KUKA KRL program: DESPA - KR 470-2 PA.src, DESPA - KR 470-2 PA.dat

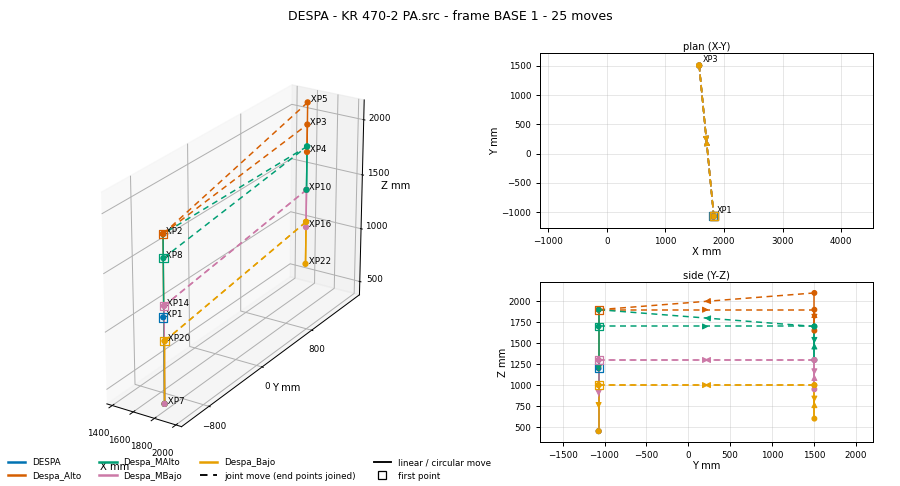
[picture p0: tool path of DESPA - KR 470-2 PA.src in frame BASE 1, 25 of 25 moves have a stored position in this frame; points joined in program order, loops and branches not executed]
--- DESPA - KR 470-2 PA.src ---
&ACCESS RVP
&REL 5
&PARAM TEMPLATE = C:\KRC\ROBOTER\TEMPLATE\vorgabe
&PARAM EDITMASK = *
DEF DESPA - KR 470-2 PA( )
;FOLD INI;%{PE}%V3.2.0,%MKUKATPBASIS,%CINIT,%VCOMMON,%P
;FOLD BAS INI;%{E}%V3.2.0,%MKUKATPBASIS,%CINIT,%VINIT,%P
GLOBAL INTERRUPT DECL 3 WHEN $STOPMESS==TRUE DO IR_STOPM ( )
INTERRUPT ON 3
BAS (#INITMOV,0 )
;ENDFOLD (BAS INI)
;FOLD A20 INI;%{E}%V3.2.0,%MKUKATPA20,%CINIT,%VINIT,%P
IF ARC20==TRUE THEN
A20 (ARC_INI)
INTERRUPT DECL 6 WHEN $CYCFLAG[3]==FALSE DO A20(TECH_STOP2)
ENDIF
;ENDFOLD (A20 INI)
;FOLD A10 INI;%{E}%V3.2.0,%MKUKATPARC,%CINIT,%VINIT,%P
IF A10_OPTION==#ACTIVE THEN
INTERRUPT DECL 4 WHEN $CYCFLAG[2]==FALSE DO A10 (#APPL_ERROR)
INTERRUPT DECL 7 WHEN A_ARC_SWI==#ACTIVE DO A10 (#ARC_SEAM)
INTERRUPT DECL 5 WHEN A_FLY_ARC==TRUE DO A10 (#HPU_ARC)
INTERRUPT  ON 5
A10_INI ( )
ENDIF
;ENDFOLD (A10 INI)
;FOLD GRIPPER INI;%{E}%V3.2.0,%MKUKATPGRIPPER,%CINIT,%VINIT,%P
USER_GRP(0,DUMMY,DUMMY,GDEFAULT)
;ENDFOLD (GRIPPER INI)
;FOLD SPOT INI;%{E}%V3.2.0,%MKUKATPSPOT,%CINIT,%VINIT,%P
USERSPOT(#INIT)
;ENDFOLD (SPOT INI)
;FOLD TOUCHSENSE INI;%{E}%V3.2.0,%MKUKATPTS,%CINIT,%VINIT,%P
IF H70_OPTION THEN
INTERRUPT DECL 15 WHEN $MEAS_PULSE[TOUCH_I[TOUCH_ACTIVE].IN_NR] DO H70 (6,CD0 )
INTERRUPT DECL 16 WHEN $ZERO_MOVE DO H70 (7,CD0 )
INTERRUPT DECL 17 WHEN $TECHPAR_C[FG_TOUCH,8]>0.5 DO H70 (8,CD0)
H70 (1,CD0 )
ENDIF
;ENDFOLD (TOUCHSENSE INI)
;FOLD USER INI;%{E}%V3.2.0,%MKUKATPUSER,%CINIT,%VINIT,%P
;Make your modifications here
;ENDFOLD (USER INI)
;ENDFOLD (INI)

; Layout : C:\Users\Albert\Desktop\Proy_Final\Final_V2\FINAL_V2.vcm
; Robot : KR 180 PA #3
; BASE_DATA[1] = {x 0,y 0,z 0,a 0,b 0,c 0}
; TOOL_DATA[1] = {x 0,y 0,z 0,a 0,b 0,c 0}
Despa_Alto()
;FOLD WAIT Time= 0.5 sec;%{PE}%R 4.1.6,%MKUKATPBASIS,%CWAIT,%VWAIT,%P 2:0.5
WAIT SEC 0.5
;ENDFOLD
Despa_MAlto()
;FOLD WAIT Time= 1 sec;%{PE}%R 4.1.6,%MKUKATPBASIS,%CWAIT,%VWAIT,%P 2:1
WAIT SEC 1
;ENDFOLD
Despa_MBajo()
;FOLD WAIT Time= 1 sec;%{PE}%R 4.1.6,%MKUKATPBASIS,%CWAIT,%VWAIT,%P 2:1
WAIT SEC 1
;ENDFOLD
Despa_Bajo()
;FOLD WAIT Time= 1 sec;%{PE}%R 4.1.6,%MKUKATPBASIS,%CWAIT,%VWAIT,%P 2:1
WAIT SEC 1
;ENDFOLD
;FOLD LIN P1  Vel= 2 m/s CPDAT1 Tool[1] Base[1];%{PE}%R 4.1.6,%MKUKATPBASIS,%CMOVE,%VLIN,%P 1:LIN, 2:P1, 3:, 5:2, 7:CPDAT1
$BWDSTART = FALSE
LDAT_ACT=LCPDAT1
BAS(#CP_DAT)
FDAT_ACT=FP1
BAS(#FRAMES)
BAS(#VEL_CP,2)
LIN XP1
;ENDFOLD
END

DEF Despa_Alto()
;FOLD PTP P2  Vel= 100 % PDAT1 Tool[1] Base[1];%{PE}%R 4.1.6,%MKUKATPBASIS,%CMOVE,%VPTP,%P 1:PTP, 2:P2, 3:, 5:100, 7:PDAT1
$BWDSTART = FALSE
PDAT_ACT=PPDAT1
BAS(#PTP_DAT)
FDAT_ACT=FP2
BAS(#FRAMES)
BAS(#VEL_PTP,100)
PTP XP2
;ENDFOLD
;FOLD PTP P3  Vel= 100 % PDAT2 Tool[1] Base[1];%{PE}%R 4.1.6,%MKUKATPBASIS,%CMOVE,%VPTP,%P 1:PTP, 2:P3, 3:, 5:100, 7:PDAT2
$BWDSTART = FALSE
PDAT_ACT=PPDAT2
BAS(#PTP_DAT)
FDAT_ACT=FP3
BAS(#FRAMES)
BAS(#VEL_PTP,100)
PTP XP3
;ENDFOLD
;FOLD LIN P4  Vel= 2 m/s CPDAT2 Tool[1] Base[1];%{PE}%R 4.1.6,%MKUKATPBASIS,%CMOVE,%VLIN,%P 1:LIN, 2:P4, 3:, 5:2, 7:CPDAT2
$BWDSTART = FALSE
LDAT_ACT=LCPDAT2
BAS(#CP_DAT)
FDAT_ACT=FP4
BAS(#FRAMES)
BAS(#VEL_CP,2)
LIN XP4
;ENDFOLD
;FOLD LIN P5  Vel= 2 m/s CPDAT3 Tool[1] Base[1];%{PE}%R 4.1.6,%MKUKATPBASIS,%CMOVE,%VLIN,%P 1:LIN, 2:P5, 3:, 5:2, 7:CPDAT3
$BWDSTART = FALSE
LDAT_ACT=LCPDAT3
BAS(#CP_DAT)
FDAT_ACT=FP5
BAS(#FRAMES)
BAS(#VEL_CP,2)
LIN XP5
;ENDFOLD
;FOLD PTP P6  Vel= 100 % PDAT3 Tool[1] Base[1];%{PE}%R 4.1.6,%MKUKATPBASIS,%CMOVE,%VPTP,%P 1:PTP, 2:P6, 3:, 5:100, 7:PDAT3
$BWDSTART = FALSE
PDAT_ACT=PPDAT3
BAS(#PTP_DAT)
FDAT_ACT=FP6
BAS(#FRAMES)
BAS(#VEL_PTP,100)
PTP XP6
;ENDFOLD
;FOLD LIN P7  Vel= 2 m/s CPDAT4 Tool[1] Base[1];%{PE}%R 4.1.6,%MKUKATPBASIS,%CMOVE,%VLIN,%P 1:LIN, 2:P7, 3:, 5:2, 7:CPDAT4
$BWDSTART = FALSE
LDAT_ACT=LCPDAT4
BAS(#CP_DAT)
FDAT_ACT=FP7
BAS(#FRAMES)
BAS(#VEL_CP,2)
LIN XP7
;ENDFOLD
END

DEF Despa_MAlto()
;FOLD PTP P8  Vel= 100 % PDAT4 Tool[1] Base[1];%{PE}%R 4.1.6,%MKUKATPBASIS,%CMOVE,%VPTP,%P 1:PTP, 2:P8, 3:, 5:100, 7:PDAT4
$BWDSTART = FALSE
PDAT_ACT=PPDAT4
BAS(#PTP_DAT)
FDAT_ACT=FP8
BAS(#FRAMES)
BAS(#VEL_PTP,100)
PTP XP8
;ENDFOLD
;FOLD PTP P9  Vel= 100 % PDAT5 Tool[1] Base[1];%{PE}%R 4.1.6,%MKUKATPBASIS,%CMOVE,%VPTP,%P 1:PTP, 2:P9, 3:, 5:100, 7:PDAT5
$BWDSTART = FALSE
PDAT_ACT=PPDAT5
BAS(#PTP_DAT)
FDAT_ACT=FP9
BAS(#FRAMES)
BAS(#VEL_PTP,100)
PTP XP9
;ENDFOLD
;FOLD LIN P10  Vel= 2 m/s CPDAT5 Tool[1] Base[1];%{PE}%R 4.1.6,%MKUKATPBASIS,%CMOVE,%VLIN,%P 1:LIN, 2:P10, 3:, 5:2, 7:CPDAT5
$BWDSTART = FALSE
LDAT_ACT=LCPDAT5
BAS(#CP_DAT)
FDAT_ACT=FP10
BAS(#FRAMES)
BAS(#VEL_CP,2)
LIN XP10
;ENDFOLD
;FOLD LIN P11  Vel= 2 m/s CPDAT6 Tool[1] Base[1];%{PE}%R 4.1.6,%MKUKATPBASIS,%CMOVE,%VLIN,%P 1:LIN, 2:P11, 3:, 5:2, 7:CPDAT6
$BWDSTART = FALSE
LDAT_ACT=LCPDAT6
BAS(#CP_DAT)
FDAT_ACT=FP11
BAS(#FRAMES)
BAS(#VEL_CP,2)
LIN XP11
;ENDFOLD
;FOLD PTP P12  Vel= 100 % PDAT6 Tool[1] Base[1];%{PE}%R 4.1.6,%MKUKATPBASIS,%CMOVE,%VPTP,%P 1:PTP, 2:P12, 3:, 5:100, 7:PDAT6
$BWDSTART = FALSE
PDAT_ACT=PPDAT6
BAS(#PTP_DAT)
FDAT_ACT=FP12
BAS(#FRAMES)
BAS(#VEL_PTP,100)
PTP XP12
;ENDFOLD
;FOLD LIN P13  Vel= 2 m/s CPDAT7 Tool[1] Base[1];%{PE}%R 4.1.6,%MKUKATPBASIS,%CMOVE,%VLIN,%P 1:LIN, 2:P13, 3:, 5:2, 7:CPDAT7
$BWDSTART = FALSE
LDAT_ACT=LCPDAT7
BAS(#CP_DAT)
FDAT_ACT=FP13
BAS(#FRAMES)
BAS(#VEL_CP,2)
LIN XP13
;ENDFOLD
END

DEF Despa_MBajo()
;FOLD PTP P14  Vel= 100 % PDAT7 Tool[1] Base[1];%{PE}%R 4.1.6,%MKUKATPBASIS,%CMOVE,%VPTP,%P 1:PTP, 2:P14, 3:, 5:100, 7:PDAT7
$BWDSTART = FALSE
PDAT_ACT=PPDAT7
BAS(#PTP_DAT)
FDAT_ACT=FP14
BAS(#FRAMES)
BAS(#VEL_PTP,100)
PTP XP14
;ENDFOLD
;FOLD PTP P15  Vel= 100 % PDAT8 Tool[1] Base[1];%{PE}%R 4.1.6,%MKUKATPBASIS,%CMOVE,%VPTP,%P 1:PTP, 2:P15, 3:, 5:100, 7:PDAT8
$BWDSTART = FALSE
PDAT_ACT=PPDAT8
BAS(#PTP_DAT)
FDAT_ACT=FP15
BAS(#FRAMES)
BAS(#VEL_PTP,100)
PTP XP15
;ENDFOLD
;FOLD LIN P16  Vel= 2 m/s CPDAT8 Tool[1] Base[1];%{PE}%R 4.1.6,%MKUKATPBASIS,%CMOVE,%VLIN,%P 1:LIN, 2:P16, 3:, 5:2, 7:CPDAT8
$BWDSTART = FALSE
LDAT_ACT=LCPDAT8
BAS(#CP_DAT)
FDAT_ACT=FP16
BAS(#FRAMES)
BAS(#VEL_CP,2)
LIN XP16
;ENDFOLD
;FOLD LIN P17  Vel= 2 m/s CPDAT9 Tool[1] Base[1];%{PE}%R 4.1.6,%MKUKATPBASIS,%CMOVE,%VLIN,%P 1:LIN, 2:P17, 3:, 5:2, 7:CPDAT9
$BWDSTART = FALSE
LDAT_ACT=LCPDAT9
BAS(#CP_DAT)
FDAT_ACT=FP17
BAS(#FRAMES)
BAS(#VEL_CP,2)
LIN XP17
;ENDFOLD
;FOLD PTP P18  Vel= 100 % PDAT9 Tool[1] Base[1];%{PE}%R 4.1.6,%MKUKATPBASIS,%CMOVE,%VPTP,%P 1:PTP, 2:P18, 3:, 5:100, 7:PDAT9
$BWDSTART = FALSE
PDAT_ACT=PPDAT9
BAS(#PTP_DAT)
FDAT_ACT=FP18
BAS(#FRAMES)
BAS(#VEL_PTP,100)
PTP XP18
;ENDFOLD
;FOLD LIN P19  Vel= 2 m/s CPDAT10 Tool[1] Base[1];%{PE}%R 4.1.6,%MKUKATPBASIS,%CMOVE,%VLIN,%P 1:LIN, 2:P19, 3:, 5:2, 7:CPDAT10
$BWDSTART = FALSE
LDAT_ACT=LCPDAT10
BAS(#CP_DAT)
FDAT_ACT=FP19
BAS(#FRAMES)
BAS(#VEL_CP,2)
LIN XP19
;ENDFOLD
END

DEF Despa_Bajo()
;FOLD PTP P20  Vel= 100 % PDAT10 Tool[1] Base[1];%{PE}%R 4.1.6,%MKUKATPBASIS,%CMOVE,%VPTP,%P 1:PTP, 2:P20, 3:, 5:100, 7:PDAT10
$BWDSTART = FALSE
PDAT_ACT=PPDAT10
BAS(#PTP_DAT)
FDAT_ACT=FP20
BAS(#FRAMES)
BAS(#VEL_PTP,100)
PTP XP20
;ENDFOLD
;FOLD PTP P21  Vel= 100 % PDAT11 Tool[1] Base[1];%{PE}%R 4.1.6,%MKUKATPBASIS,%CMOVE,%VPTP,%P 1:PTP, 2:P21, 3:, 5:100, 7:PDAT11
$BWDSTART = FALSE
PDAT_ACT=PPDAT11
BAS(#PTP_DAT)
FDAT_ACT=FP21
BAS(#FRAMES)
BAS(#VEL_PTP,100)
PTP XP21
;ENDFOLD
;FOLD LIN P22  Vel= 2 m/s CPDAT11 Tool[1] Base[1];%{PE}%R 4.1.6,%MKUKATPBASIS,%CMOVE,%VLIN,%P 1:LIN, 2:P22, 3:, 5:2, 7:CPDAT11
$BWDSTART = FALSE
LDAT_ACT=LCPDAT11
BAS(#CP_DAT)
FDAT_ACT=FP22
BAS(#FRAMES)
BAS(#VEL_CP,2)
LIN XP22
;ENDFOLD
;FOLD LIN P23  Vel= 2 m/s CPDAT12 Tool[1] Base[1];%{PE}%R 4.1.6,%MKUKATPBASIS,%CMOVE,%VLIN,%P 1:LIN, 2:P23, 3:, 5:2, 7:CPDAT12
$BWDSTART = FALSE
LDAT_ACT=LCPDAT12
BAS(#CP_DAT)
FDAT_ACT=FP23
BAS(#FRAMES)
BAS(#VEL_CP,2)
LIN XP23
;ENDFOLD
;FOLD PTP P24  Vel= 100 % PDAT12 Tool[1] Base[1];%{PE}%R 4.1.6,%MKUKATPBASIS,%CMOVE,%VPTP,%P 1:PTP, 2:P24, 3:, 5:100, 7:PDAT12
$BWDSTART = FALSE
PDAT_ACT=PPDAT12
BAS(#PTP_DAT)
FDAT_ACT=FP24
BAS(#FRAMES)
BAS(#VEL_PTP,100)
PTP XP24
;ENDFOLD
;FOLD LIN P25  Vel= 2 m/s CPDAT13 Tool[1] Base[1];%{PE}%R 4.1.6,%MKUKATPBASIS,%CMOVE,%VLIN,%P 1:LIN, 2:P25, 3:, 5:2, 7:CPDAT13
$BWDSTART = FALSE
LDAT_ACT=LCPDAT13
BAS(#CP_DAT)
FDAT_ACT=FP25
BAS(#FRAMES)
BAS(#VEL_CP,2)
LIN XP25
;ENDFOLD
END

--- DESPA - KR 470-2 PA.dat ---
&ACCESS RVP
&REL 5
&PARAM TEMPLATE = C:\KRC\ROBOTER\TEMPLATE\vorgabe
&PARAM EDITMASK = *
DEFDAT  despa - kr 470-2 pa
;FOLD EXTERNAL DECLARATIONS;%{PE}%V3.2.0,%MKUKATPBASIS,%CEXT,%VCOMMON,%P
;FOLD BAS EXT;%{PE}%V3.2.0,%MKUKATPBASIS,%CEXT,%VEXT,%P
EXT  BAS (BAS_COMMAND  :IN,REAL  :IN )
DECL INT SUCCESS
;ENDFOLD
;FOLD A10 EXT;%{E}%V3.2.0,%MKUKATPARC,%CEXT,%VEXT,%P
EXT  A10 (A_CMD_T  :IN,A_STRT_T  :IN,A_WELD_T  :IN,A_END_T  :IN,INT  :IN )
;ENDFOLD
;FOLD A20 EXT;%{E}%V3.2.0,%MKUKATPA20,%CEXT,%VEXT,%P
EXT  A20 (INT  :IN,WELD_ST  :IN,WELD_FI  :IN,INT  :IN )
;ENDFOLD
;FOLD GRIPPER EXT;%{E}%V3.2.0,%MKUKATPGRIPPER,%CEXT,%VEXT,%P
EXT  H50 (INT  :IN,INT  :IN,INT  :IN,GRP_TYP  :IN )
;ENDFOLD
;FOLD SPOT EXT;%{E}%V3.2.0,%MKUKATPSPOT,%CEXT,%VEXT,%P
EXT  USERSPOT (S_COMMAND  :IN,SPOT_TYPE  :IN )
;ENDFOLD
;FOLD TOUCHSENSE EXT;%{E}%V3.2.0,%MKUKATPTS,%CEXT,%VEXT,%P
EXT  H70 (INT  :IN,SRCH_TYP_2  :OUT,E6POS  :IN,SRCH_TYP_3  :IN,SRCH_TYP_2  :IN,SRCH_TYP_2  :IN,SRCH_TYP_2  :IN,SRCH_TYP_2  :IN,SRCH_TYP_2  :IN,INT  :IN )
;ENDFOLD
;FOLD USER EXT;%{E}%V3.2.0,%MKUKATPUSER,%CEXT,%VEXT,%P
;Make here your modifications
;ENDFOLD
;ENDFOLD

DECL E6POS XP1={x 1815.4,y -1070.28,z 1200,a -90,b 0,c -180,s 2,t 2,e1 0,e2 0,e3 0,e4 0,e5 0,e6 0}
DECL FDAT FP1={TOOL_NO 1,BASE_NO 1,IPO_FRAME #BASE}
DECL LDAT LCPDAT1={VEL 2.0,ACC 100.0,APO_DIST 100.0,APO_FAC 50.0}
DECL E6POS XP2={x 1825.4,y -1070.28,z 1900,a 90,b -180,c 0,s 2,t 2,e1 0,e2 0,e3 0,e4 0,e5 0,e6 0}
DECL FDAT FP2={TOOL_NO 1,BASE_NO 1,IPO_FRAME #BASE}
DECL PDAT PPDAT1={VEL 100.0,ACC 100.0,APO_DIST 100.0}
DECL E6POS XP3={x 1575.4,y 1504.72,z 1900,a 0,b 180,c 0,s 2,t 35,e1 0,e2 0,e3 0,e4 0,e5 0,e6 0}
DECL FDAT FP3={TOOL_NO 1,BASE_NO 1,IPO_FRAME #BASE}
DECL PDAT PPDAT2={VEL 100.0,ACC 100.0,APO_DIST 100.0}
DECL E6POS XP4={x 1575.4,y 1504.72,z 1650,a 0,b 180,c 0,s 2,t 35,e1 0,e2 0,e3 0,e4 0,e5 0,e6 0}
DECL FDAT FP4={TOOL_NO 1,BASE_NO 1,IPO_FRAME #BASE}
DECL LDAT LCPDAT2={VEL 2.0,ACC 100.0,APO_DIST 100.0,APO_FAC 50.0}
DECL E6POS XP5={x 1575.4,y 1504.72,z 2100,a 0,b 180,c 0,s 2,t 35,e1 0,e2 0,e3 0,e4 0,e5 0,e6 0}
DECL FDAT FP5={TOOL_NO 1,BASE_NO 1,IPO_FRAME #BASE}
DECL LDAT LCPDAT3={VEL 2.0,ACC 100.0,APO_DIST 100.0,APO_FAC 50.0}
DECL E6POS XP6={x 1825.4,y -1070.28,z 1900,a 90,b 180,c 0,s 2,t 2,e1 0,e2 0,e3 0,e4 0,e5 0,e6 0}
DECL FDAT FP6={TOOL_NO 1,BASE_NO 1,IPO_FRAME #BASE}
DECL PDAT PPDAT3={VEL 100.0,ACC 100.0,APO_DIST 100.0}
DECL E6POS XP7={x 1815.4,y -1070.28,z 450,a -90,b 0,c 180,s 2,t 2,e1 0,e2 0,e3 0,e4 0,e5 0,e6 0}
DECL FDAT FP7={TOOL_NO 1,BASE_NO 1,IPO_FRAME #BASE}
DECL LDAT LCPDAT4={VEL 2.0,ACC 100.0,APO_DIST 100.0,APO_FAC 50.0}
DECL E6POS XP8={x 1825.4,y -1070.28,z 1700,a 90,b -180,c 0,s 2,t 2,e1 0,e2 0,e3 0,e4 0,e5 0,e6 0}
DECL FDAT FP8={TOOL_NO 1,BASE_NO 1,IPO_FRAME #BASE}
DECL PDAT PPDAT4={VEL 100.0,ACC 100.0,APO_DIST 100.0}
DECL E6POS XP9={x 1575.4,y 1504.72,z 1700,a 0,b 180,c 0,s 2,t 35,e1 0,e2 0,e3 0,e4 0,e5 0,e6 0}
DECL FDAT FP9={TOOL_NO 1,BASE_NO 1,IPO_FRAME #BASE}
DECL PDAT PPDAT5={VEL 100.0,ACC 100.0,APO_DIST 100.0}
DECL E6POS XP10={x 1575.4,y 1504.72,z 1300,a 0,b 180,c 0,s 2,t 35,e1 0,e2 0,e3 0,e4 0,e5 0,e6 0}
DECL FDAT FP10={TOOL_NO 1,BASE_NO 1,IPO_FRAME #BASE}
DECL LDAT LCPDAT5={VEL 2.0,ACC 100.0,APO_DIST 100.0,APO_FAC 50.0}
DECL E6POS XP11={x 1575.4,y 1504.72,z 1700,a 0,b 180,c 0,s 2,t 35,e1 0,e2 0,e3 0,e4 0,e5 0,e6 0}
DECL FDAT FP11={TOOL_NO 1,BASE_NO 1,IPO_FRAME #BASE}
DECL LDAT LCPDAT6={VEL 2.0,ACC 100.0,APO_DIST 100.0,APO_FAC 50.0}
DECL E6POS XP12={x 1825.4,y -1070.28,z 1900,a 90,b 180,c 0,s 2,t 2,e1 0,e2 0,e3 0,e4 0,e5 0,e6 0}
DECL FDAT FP12={TOOL_NO 1,BASE_NO 1,IPO_FRAME #BASE}
DECL PDAT PPDAT6={VEL 100.0,ACC 100.0,APO_DIST 100.0}
DECL E6POS XP13={x 1815.4,y -1070.28,z 450,a -90,b 0,c -180,s 2,t 2,e1 0,e2 0,e3 0,e4 0,e5 0,e6 0}
DECL FDAT FP13={TOOL_NO 1,BASE_NO 1,IPO_FRAME #BASE}
DECL LDAT LCPDAT7={VEL 2.0,ACC 100.0,APO_DIST 100.0,APO_FAC 50.0}
DECL E6POS XP14={x 1825.4,y -1070.28,z 1300,a 90,b -180,c 0,s 2,t 2,e1 0,e2 0,e3 0,e4 0,e5 0,e6 0}
DECL FDAT FP14={TOOL_NO 1,BASE_NO 1,IPO_FRAME #BASE}
DECL PDAT PPDAT7={VEL 100.0,ACC 100.0,APO_DIST 100.0}
DECL E6POS XP15={x 1575.4,y 1504.72,z 1300,a 0,b 180,c 0,s 2,t 35,e1 0,e2 0,e3 0,e4 0,e5 0,e6 0}
DECL FDAT FP15={TOOL_NO 1,BASE_NO 1,IPO_FRAME #BASE}
DECL PDAT PPDAT8={VEL 100.0,ACC 100.0,APO_DIST 100.0}
DECL E6POS XP16={x 1575.4,y 1504.72,z 950,a 0,b 180,c 0,s 2,t 35,e1 0,e2 0,e3 0,e4 0,e5 0,e6 0}
DECL FDAT FP16={TOOL_NO 1,BASE_NO 1,IPO_FRAME #BASE}
DECL LDAT LCPDAT8={VEL 2.0,ACC 100.0,APO_DIST 100.0,APO_FAC 50.0}
DECL E6POS XP17={x 1575.4,y 1504.72,z 1300,a 0,b 180,c 0,s 2,t 35,e1 0,e2 0,e3 0,e4 0,e5 0,e6 0}
DECL FDAT FP17={TOOL_NO 1,BASE_NO 1,IPO_FRAME #BASE}
DECL LDAT LCPDAT9={VEL 2.0,ACC 100.0,APO_DIST 100.0,APO_FAC 50.0}
DECL E6POS XP18={x 1825.4,y -1070.28,z 1300,a 90,b 180,c 0,s 2,t 2,e1 0,e2 0,e3 0,e4 0,e5 0,e6 0}
DECL FDAT FP18={TOOL_NO 1,BASE_NO 1,IPO_FRAME #BASE}
DECL PDAT PPDAT9={VEL 100.0,ACC 100.0,APO_DIST 100.0}
DECL E6POS XP19={x 1815.4,y -1070.28,z 450,a -90,b 0,c -180,s 2,t 2,e1 0,e2 0,e3 0,e4 0,e5 0,e6 0}
DECL FDAT FP19={TOOL_NO 1,BASE_NO 1,IPO_FRAME #BASE}
DECL LDAT LCPDAT10={VEL 2.0,ACC 100.0,APO_DIST 100.0,APO_FAC 50.0}
DECL E6POS XP20={x 1825.4,y -1070.28,z 1000,a 90,b 180,c 0,s 2,t 2,e1 0,e2 0,e3 0,e4 0,e5 0,e6 0}
DECL FDAT FP20={TOOL_NO 1,BASE_NO 1,IPO_FRAME #BASE}
DECL PDAT PPDAT10={VEL 100.0,ACC 100.0,APO_DIST 100.0}
DECL E6POS XP21={x 1575.4,y 1504.72,z 1000,a 0,b 180,c 0,s 2,t 35,e1 0,e2 0,e3 0,e4 0,e5 0,e6 0}
DECL FDAT FP21={TOOL_NO 1,BASE_NO 1,IPO_FRAME #BASE}
DECL PDAT PPDAT11={VEL 100.0,ACC 100.0,APO_DIST 100.0}
DECL E6POS XP22={x 1575.4,y 1504.72,z 600,a 0,b 180,c 0,s 2,t 35,e1 0,e2 0,e3 0,e4 0,e5 0,e6 0}
DECL FDAT FP22={TOOL_NO 1,BASE_NO 1,IPO_FRAME #BASE}
DECL LDAT LCPDAT11={VEL 2.0,ACC 100.0,APO_DIST 100.0,APO_FAC 50.0}
DECL E6POS XP23={x 1575.4,y 1504.72,z 1000,a 0,b 180,c 0,s 2,t 35,e1 0,e2 0,e3 0,e4 0,e5 0,e6 0}
DECL FDAT FP23={TOOL_NO 1,BASE_NO 1,IPO_FRAME #BASE}
DECL LDAT LCPDAT12={VEL 2.0,ACC 100.0,APO_DIST 100.0,APO_FAC 50.0}
DECL E6POS XP24={x 1825.4,y -1070.28,z 1000,a 90,b 180,c 0,s 2,t 2,e1 0,e2 0,e3 0,e4 0,e5 0,e6 0}
DECL FDAT FP24={TOOL_NO 1,BASE_NO 1,IPO_FRAME #BASE}
DECL PDAT PPDAT12={VEL 100.0,ACC 100.0,APO_DIST 100.0}
DECL E6POS XP25={x 1815.4,y -1070.28,z 450,a -90,b 0,c -180,s 2,t 2,e1 0,e2 0,e3 0,e4 0,e5 0,e6 0}
DECL FDAT FP25={TOOL_NO 1,BASE_NO 1,IPO_FRAME #BASE}
DECL LDAT LCPDAT13={VEL 2.0,ACC 100.0,APO_DIST 100.0,APO_FAC 50.0}
ENDDAT
